FUNCTION_BLOCK FB_Env
(*
	The environment should provide methods like step, reset etc...
	If the environment is outside of the PLC environment, it should act like a proxy, or contact one
*)
VAR_INPUT
END_VAR
VAR_OUTPUT
	bResetEnvironmentOK : BOOL;
	bStartProxyOK : BOOL;
	bEnvStepRequestedOK : BOOL;
	state : INT;
	newState : INT;
	reward : INT;
	done : BOOL;
END_VAR
VAR
	_bEnvResetRequested : BOOL;
	_bProxyStarted : BOOL;
	_bEnvStepRequested : BOOL;
	_bStopEnvironmentRequested : BOOL;
	_actionToTake : INT;
	startProxy : NT_StartProcess;
	sPathToBatchFile : STRING;
	sPathToBatchFileFolder : STRING;
END_VAR

startProxy(
	NETID:= '', 
	PATHSTR:= sPathToBatchFile, 
	DIRNAME:= sPathToBatchFileFolder, 
	COMNDLINE:= , 
	START:= FALSE, 
	TMOUT:= , 
	BUSY=> , 
	ERR=> , 
	ERRID=> );

METHOD M_ConfirmEnvResetRead
VAR_INPUT
END_VAR
bResetEnvironmentOK := FALSE;
_bEnvResetRequested := FALSE;
END_METHOD

METHOD M_ConfirmEnvStepRequestRead
VAR_INPUT
END_VAR
bEnvStepRequestedOK := FALSE;
_bEnvStepRequested := FALSE;
END_METHOD

METHOD PUBLIC M_ResetEnvironment
VAR_INPUT
END_VAR
IF NOT _bEnvResetRequested THEN
	_bEnvResetRequested := TRUE;
END_IF
END_METHOD

METHOD M_ResetInternalStates
VAR_INPUT
END_VAR
bResetEnvironmentOK := FALSE;
bStartProxyOK := FALSE;
bEnvStepRequestedOK := FALSE;
done := FALSE;
_bEnvResetRequested := FALSE;
_bEnvStepRequested := FALSE;
END_METHOD

METHOD PUBLIC M_StartProxy : BOOL
VAR_INPUT
END_VAR
IF NOT _bProxyStarted THEN
	_bProxyStarted := TRUE;
	startProxy(
		NETID:= '', 
		PATHSTR:= sPathToBatchFile, 
		DIRNAME:= sPathToBatchFileFolder, 
		COMNDLINE:= , 
		START:= TRUE, 
		TMOUT:= , 
		BUSY=> , 
		ERR=> , 
		ERRID=> );
END_IF
END_METHOD

METHOD M_Step 
VAR_INPUT
	actionToTake : INT;
END_VAR
IF NOT _bEnvStepRequested THEN
	_actionToTake := actionToTake;
	_bEnvStepRequested := TRUE;
END_IF
END_METHOD

METHOD M_StopEnvironment
VAR_INPUT
END_VAR
IF NOT _bStopEnvironmentRequested THEN
	_bStopEnvironmentRequested := TRUE;
END_IF
END_METHOD

END_FUNCTION_BLOCK

(* stored: Version 1.1.0.1, ProductVersion 3.1.4024.12
   POU FB_Env: Id {b1c361d3-a423-4771-a6f2-cf52b12a39f5}, SpecialFunc None
   Method M_ConfirmEnvResetRead: Id {ebb2ffa5-5745-47cd-85a6-94c5fc8caad4}
   Method M_ConfirmEnvStepRequestRead: Id {894b98f3-372b-498c-83cf-8a66055ed630}
   Method M_ResetEnvironment: Id {eeca9014-46b2-4824-b207-3ec1e4c03604}
   Method M_ResetInternalStates: Id {e99c22c6-1c5b-4b89-bd0e-7768d09a3316}
   Method M_StartProxy: Id {0895a20c-0eaa-4612-ab3a-3ec5fdffe64d}
   Method M_Step: Id {e7326f5d-4df5-4679-888e-9e87b50800c0}
   Method M_StopEnvironment: Id {c0e520a0-a0bb-4a46-a4d8-ba7b016ba020} *)
